PROGRAM MAIN
VAR
END_VAR

END_PROGRAM

(* stored: Version 1.1.0.1
   POU MAIN: Id {4e545c59-324d-4331-98a3-1208180d1ff0} *)
